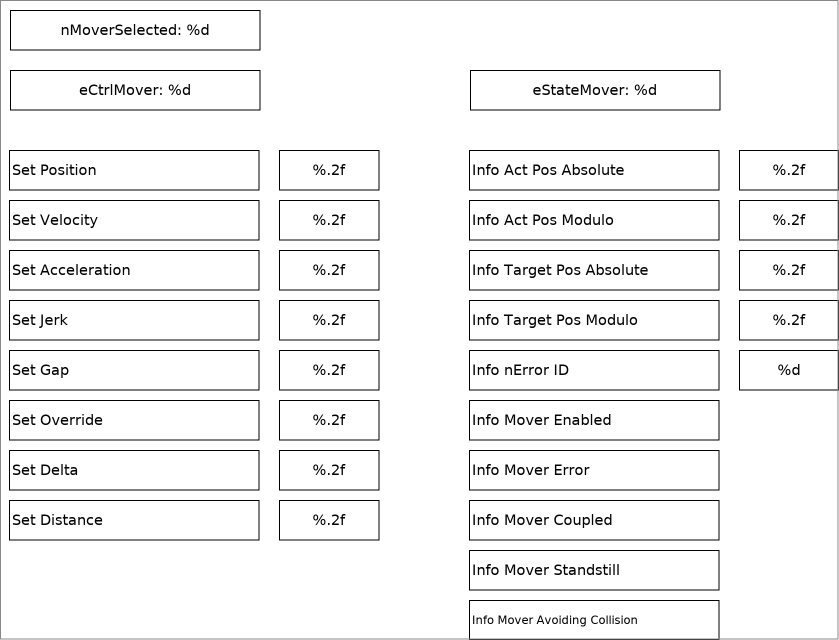
VISUALIZATION MOVER_VISU  // 839x640
    Rectangle (10,10 250x40), "nMoverSelected: %d", text variable: MOVER.nMoverSelected
        OnMouseClick: write the text variable via VisuDialogs.Numpad, min 1, max MAX_MOVER, title 'Selected Mover'
    Rectangle (10,70 250x40), "eCtrlMover: %d", text variable: MOVER.eCtrl
        OnMouseClick: write the text variable via Default, min 0, max 220, title 'Mover Command'
    Rectangle (9,150 250x40), "Set Position"
    Rectangle (9,200 250x40), "Set Velocity"
    Rectangle (9,250 250x40), "Set Acceleration"
    Rectangle (9,300 250x40), "Set Jerk"
    Rectangle (9,350 250x40), "Set Gap"
    Rectangle (9,400 250x40), "Set Override"
    Rectangle (9,450 250x40), "Set Delta"
    Rectangle (9,500 250x40), "Set Distance"
    Rectangle (279,150 100x40), "%.2f", text variable: GVL_XTS.MoveData[MOVER.nMoverSelected].rPos
        OnMouseClick: write the text variable via Default
    Rectangle (279,200 100x40), "%.2f", text variable: GVL_XTS.MoveData[MOVER.nMoverSelected].rVelo
        OnMouseClick: write the text variable via Default
    Rectangle (279,250 100x40), "%.2f", text variable: GVL_XTS.MoveData[MOVER.nMoverSelected].rAcc
        OnMouseClick: write the text variable via Default
    Rectangle (279,300 100x40), "%.2f", text variable: GVL_XTS.MoveData[MOVER.nMoverSelected].rJerk
        OnMouseClick: write the text variable via Default
    Rectangle (279,350 100x40), "%.2f", text variable: GVL_XTS.MoveData[MOVER.nMoverSelected].rGap
        OnMouseClick: write the text variable via Default
    Rectangle (279,400 100x40), "%.2f", text variable: GVL_XTS.MoveData[MOVER.nMoverSelected].rOverride
        OnMouseClick: write the text variable via Default
    Rectangle (279,450 100x40), "%.2f", text variable: GVL_XTS.MoveData[MOVER.nMoverSelected].rDelta
        OnMouseClick: write the text variable via Default
    Rectangle (279,500 100x40), "%.2f", text variable: GVL_XTS.MoveData[MOVER.nMoverSelected].rDistance
        OnMouseClick: write the text variable via Default
    Rectangle (469,150 250x40), "Info Act Pos Absolute"
    Rectangle (469,200 250x40), "Info Act Pos Modulo"
    Rectangle (469,250 250x40), "Info Target Pos Absolute"
    Rectangle (469,300 250x40), "Info Target Pos Modulo"
    Rectangle (469,350 250x40), "Info nError ID"
    Rectangle (739,150 100x40), "%.2f", text variable: GVL_XTS.MoverInfo[MOVER.nMoverSelected].rAbsActPos
    Rectangle (739,200 100x40), "%.2f", text variable: GVL_XTS.MoverInfo[MOVER.nMoverSelected].rModuloActPos
    Rectangle (739,250 100x40), "%.2f", text variable: GVL_XTS.MoverInfo[MOVER.nMoverSelected].rAbsTargetPos
    Rectangle (739,300 100x40), "%.2f", text variable: GVL_XTS.MoverInfo[MOVER.nMoverSelected].rModuloTargetPos
    Rectangle (739,350 100x40), "%d", text variable: GVL_XTS.MoverInfo[MOVER.nMoverSelected].nErrorId
    Rectangle (469,400 250x40), "Info Mover Enabled", colour toggle: GVL_XTS.MoverInfo[MOVER.nMoverSelected].bMoverEnabled
    Rectangle (469,450 250x40), "Info Mover Error", colour toggle: GVL_XTS.MoverInfo[MOVER.nMoverSelected].bMoverError
    Rectangle (469,500 250x40), "Info Mover Coupled", colour toggle: GVL_XTS.MoverInfo[MOVER.nMoverSelected].bMoverCoupled
    Rectangle (469,550 250x40), "Info Mover Standstill", colour toggle: GVL_XTS.MoverInfo[MOVER.nMoverSelected].bMoverStandstill
    Rectangle (469,600 250x40), "Info Mover Avoiding Collision", colour toggle: GVL_XTS.MoverInfo[MOVER.nMoverSelected].bMoverAvoidingCollision
    Rectangle (470,70 250x40), "eStateMover: %d", text variable: MOVER.eState
END_VISUALIZATION

(* stored: Version 1.1.0.1, ProductVersion 3.1.4024.12
   Visu MOVER_VISU: Id {c9fb373c-2482-41b3-8168-553de4317393} *)
